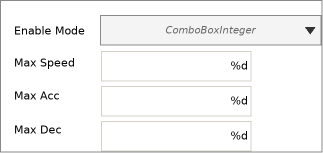
VISUALIZATION visStandardMotorSettings  // 323x153
VAR_INPUT
	refSetting : REFERENCE TO ST_StandardMotorSettings;
END_VAR
VAR CONSTANT
	cMinSpeed : UINT := 0;
	cMaxSpeed : UINT := 1000;
	cMinAcc : UINT := 1;
	cMaxAcc : UINT := 10000;
	cMinDec : UINT := 1;
	cMaxDec : UINT := 10000;
	cDialog1 : STRING := 'Max Speed in 0.1%';
	cDialog2 : STRING := 'Max Acc';
	cDialog3 : STRING := 'Max Dec';
END_VAR
    Label (11,48 150x30), "Max Speed"
    Label (11,81 150x30), "Max Acc"
    Label (11,115 150x30), "Max Dec"
    Label (11,16 150x30), "Enable Mode"
    ComboBoxInteger (100,15 221x30), variable: refSetting.eEnableMode, text list: 'txtLstMotorEnableMode'
    Textfield (101,51 150x30), "%d", text variable: refSetting.nMaxSpeed
        OnMouseClick: write the text variable via Default, min cMinSpeed, max cMaxSpeed, title cDialog1
    Textfield (101,86 150x30), "%d", text variable: refSetting.nMaxAcc
        OnMouseClick: write the text variable via Default, min cMinAcc, max cMaxAcc, title cDialog2
    Textfield (101,121 150x30), "%d", text variable: refSetting.nMaxDec
        OnMouseClick: write the text variable via Default, min cMinDec, max cMaxDec, title cDialog3
END_VISUALIZATION

(* stored: Version 1.1.0.1, ProductVersion 3.1.4019.2
   Visu visStandardMotorSettings: Id {98464449-d33c-46bd-b88d-722fa7472887} *)
